{attribute addProperty BoxType "EPP2809-0021-0016"}
{attribute addProperty Id "ChannelAT %Q*ARRAY[0..15] OF Channel_7F374EB0128160WcStateAT %I*WcState_64F6A8C6810InfoDataAT %I*InfoData_192954DE1620"}
{attribute addProperty CRC "3898205996"}
{attribute addProperty SizeInBites "152"}
{attribute addProperty SizeInBytes "19"}
TYPE EPP2809_5A2A5F29 :
STRUCT
	{attribute addProperty Name "Channel"}
	Channel : ARRAY[0..15] OF Channel_7F374EB0;
	{attribute addProperty Name "WcState"}
	WcState : WcState_64F6A8C6;
	{attribute addProperty Name "InfoData"}
	InfoData : InfoData_192954DE;
END_STRUCT
END_TYPE

(* stored: Version 1.2.0.0, ProductVersion 3.1.4024.9
   DUT EPP2809_5A2A5F29: Id {0f3655a3-d96b-4e2b-aca1-a4db4d9be77d} *)
